# EPICS alarm handler configuration: css_share/detectors/SVT/alh/SVT.R1.S2.alhConfig
GROUP NULL S2
GROUP S2 HV
GROUP HV TOP
GROUP TOP SVT-HFCB_HV_R1_M2_Top
CHANNEL SVT-HFCB_HV_R1_M2_Top B_SVT_HV_R1S2T_Slot7:outputMeasSenseVAlm
$ALIAS B_SVT_HV_R1S2T_Slot7 Measured Voltage
$STATCOMMAND HIHI caput R1S2T:MODPB_OFF 1
$STATCOMMAND LOLO caput R1S2T:MODPB_OFF 1
CHANNEL SVT-HFCB_HV_R1_M2_Top B_SVT_HV_R1S2T_Slot7:outputMeasCurrentAlm
$ALIAS B_SVT_HV_R1S2T_Slot7 Measured Current
$STATCOMMAND HIHI caput R1S2T:MODPB_OFF 1

GROUP HV BOTTOM
GROUP BOTTOM SVT-HFCB_HV_R1_M2_Bottom
CHANNEL SVT-HFCB_HV_R1_M2_Bottom B_SVT_HV_R1S2B_Slot7:outputMeasSenseVAlm
$ALIAS B_SVT_HV_R1S2B_Slot7 Measured Voltage
$STATCOMMAND HIHI caput R1S2B:MODPB_OFF 1
$STATCOMMAND LOLO caput R1S2B:MODPB_OFF 1
CHANNEL SVT-HFCB_HV_R1_M2_Bottom B_SVT_HV_R1S2B_Slot7:outputMeasCurrentAlm
$ALIAS B_SVT_HV_R1S2B_Slot7 Measured Current
$STATCOMMAND HIHI caput R1S2B:MODPB_OFF 1

GROUP S2 LV_VA
GROUP LV_VA TOP
GROUP TOP SVT-HFCB_VDDA_R1_M2_Top
CHANNEL SVT-HFCB_VDDA_R1_M2_Top B_SVT_LV_VA_R1S2T_Slot1:outputMeasSenseVAlm
$ALIAS B_SVT_LV_VA_R1S2T_Slot1 Measured Voltage
$STATCOMMAND HIHI caput R1S2T:MODPB_OFF 1
$STATCOMMAND LOLO caput R1S2T:MODPB_OFF 1
CHANNEL SVT-HFCB_VDDA_R1_M2_Top B_SVT_LV_VA_R1S2T_Slot1:outputMeasCurrentAlm
$ALIAS B_SVT_LV_VA_R1S2T_Slot1 Measured Current
$STATCOMMAND HIHI caput R1S2T:MODPB_OFF 1

GROUP LV_VA BOTTOM
GROUP BOTTOM SVT-HFCB_VDDA_R1_M2_Bottom
CHANNEL SVT-HFCB_VDDA_R1_M2_Bottom B_SVT_LV_VA_R1S2B_Slot1:outputMeasSenseVAlm
$ALIAS B_SVT_LV_VA_R1S2B_Slot1 Measured Voltage
$STATCOMMAND HIHI caput R1S2B:MODPB_OFF 1
$STATCOMMAND LOLO caput R1S2B:MODPB_OFF 1
CHANNEL SVT-HFCB_VDDA_R1_M2_Bottom B_SVT_LV_VA_R1S2B_Slot1:outputMeasCurrentAlm
$ALIAS B_SVT_LV_VA_R1S2B_Slot1 Measured Current
$STATCOMMAND HIHI caput R1S2B:MODPB_OFF 1

GROUP S2 LV_VD
GROUP LV_VD TOP
GROUP TOP SVT-HFCB_VDDD_R1_M2_Top
CHANNEL SVT-HFCB_VDDD_R1_M2_Top B_SVT_LV_VD_R1S2T_Slot1:outputMeasSenseVAlm
$ALIAS B_SVT_LV_VD_R1S2T_Slot1 Measured Voltage
$STATCOMMAND HIHI caput R1S2T:MODPB_OFF 1
$STATCOMMAND LOLO caput R1S2T:MODPB_OFF 1
CHANNEL SVT-HFCB_VDDD_R1_M2_Top B_SVT_LV_VD_R1S2T_Slot1:outputMeasCurrentAlm
$ALIAS B_SVT_LV_VD_R1S2T_Slot1 Measured Current
$STATCOMMAND HIHI caput R1S2T:MODPB_OFF 1

GROUP LV_VD BOTTOM
GROUP BOTTOM SVT-HFCB_VDDD_R1_M2_Bottom
CHANNEL SVT-HFCB_VDDD_R1_M2_Bottom B_SVT_LV_VD_R1S2B_Slot1:outputMeasSenseVAlm
$ALIAS B_SVT_LV_VD_R1S2B_Slot1 Measured Voltage
$STATCOMMAND HIHI caput R1S2B:MODPB_OFF 1
$STATCOMMAND LOLO caput R1S2B:MODPB_OFF 1
CHANNEL SVT-HFCB_VDDD_R1_M2_Bottom B_SVT_LV_VD_R1S2B_Slot1:outputMeasCurrentAlm
$ALIAS B_SVT_LV_VD_R1S2B_Slot1 Measured Current
$STATCOMMAND HIHI caput R1S2B:MODPB_OFF 1

GROUP S2 TEMP
GROUP TEMP TOP
CHANNEL TOP B_SVT_TEMP_R1S2T_Slot2Alm
$ALIAS SVT-HFCB_Temp_R1_M2_Top Temperature
$STATCOMMAND HIHI caput R1S2T:MODPB_OFF 1
$STATCOMMAND LOLO caput R1S2T:MODPB_OFF 1

GROUP TEMP BOTTOM
CHANNEL BOTTOM B_SVT_TEMP_R1S2B_Slot2Alm
$ALIAS SVT-HFCB_Temp_R1_M2_Bottom Temperature
$STATCOMMAND HIHI caput R1S2B:MODPB_OFF 1
$STATCOMMAND LOLO caput R1S2B:MODPB_OFF 1
